PROGRAM P_MyLight_Test_CFC
VAR
	fbMyLight			:	FB_MyLight1;
	bOn					:	BOOL;
	bOff				:	BOOL;
	bRecallMinLevel		:	BOOL;
	bSetControlLevel	:	BOOL;
	nSetControlLevel	:	BYTE;
	bControlLevel		:	BOOL;
	nControlLevel		:	BYTE;
END_VAR

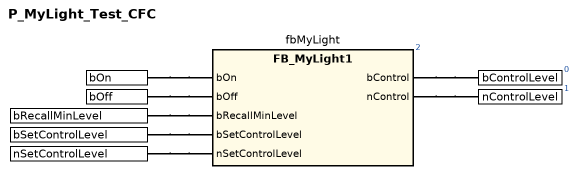
bControlLevel := fbMyLight.bControl;
nControlLevel := fbMyLight.nControl;
fbMyLight(
    bOn := bOn,
    bOff := bOff,
    bRecallMinLevel := bRecallMinLevel,
    bSetControlLevel := bSetControlLevel,
    nSetControlLevel := nSetControlLevel); // FB_MyLight1

END_PROGRAM

(* stored: Version 1.1.0.1, ProductVersion 3.1.4024.12
   POU P_MyLight_Test_CFC: Id {d3b75a9e-a061-47a8-b747-b803b819562c}, SpecialFunc None *)
